TYPE Serial_FunctionResult :
(
	NO_ERROR := -1,
	BUSY := 0,
	COM_UNKNOWN_CHANNEL,
	COM_IO_CONTROL_ERROR,
	COM_SEND_ERROR,
	COM_RECEIVE_ERROR,
	COM_NO_STRING_RECEIVED
);
END_TYPE

(* stored: Version 1.1.0.1, ProductVersion 3.1.0.36
   DUT Serial_FunctionResult: Id {efeefaa8-8328-4963-9178-ab7055e98609} *)
